{attribute 'qualified_only'}
VAR_GLOBAL
	StateManager : StateManager;
	iJogButton AT %I* : BOOL;	
	oJogButtonLight AT %Q* : BOOL;
	
	ioADSRead : FB_ReadADSSymByName;	
	ioADSWrite	: FB_WriteADSSymByName;
END_VAR

(* stored: Version 1.1.0.1, ProductVersion 3.1.4022.11
   GVL Cell: Id {2a2bb7cf-df64-47af-9771-33b156960614} *)
